FUNCTION Convert_LINT_TO_ULINT : Hresult
VAR_INPUT
	in : LINT;
	out : REFERENCE TO ULINT;
END_VAR
VAR
	converted : ULINT;
END_VAR

converted := LINT_TO_ULINT(in);

IF (ULINT_TO_LINT(converted) <> in) THEN
	Convert_LINT_TO_ULINT := INCOMPATIBLE;
	RETURN;
END_IF

out := converted;

END_FUNCTION

(* stored: Version 1.1.0.1, ProductVersion 3.1.4024.12
   POU Convert_LINT_TO_ULINT: Id {3f0f34cf-c443-480d-b9da-3b88e28ef0b5}, SpecialFunc None *)
